{attribute 'qualified_only'}
VAR_GLOBAL CONSTANT
	AlarmListSize	: DINT := 50;
END_VAR

(* stored: Version 1.1.0.1
   GVL Param_SupervisorBase: Id {9e4f26f4-016c-4a44-95f1-563266ae90c3}, ParameterList True *)
